ABB RobotStudio station: ABBPingPongRobot.rspag

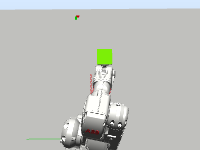
--- station ---
Station ABBPingPongRobot (saved by RobotStudio 6.8.8148.134)
Controller IRB_140_6kg_0.81m
  mechanical unit ROB_1: IRB140_6_81_C_03, 6 joints, base frame (0, 0, 0) mm
Layout (positions relative to the parent item):
  - IRB140_6_81_C_03 [mechanism, from Robots\IRB140_6_81_C_G_03.rslib] at (0, 0, 0) mm; joint values [-0.2001, 0.5892, 0.304, 2.8895, 0.9078, -2.9944] (rad or m)
  - PingPongTool [part] at (563.14, -101.19, 355.17) mm, rotated rx -95.85 ry 89.44 rz -95.98 deg
Attachment: PingPongTool is attached to IRB140_6_81_C_03 / Link6
Targets, tools, work objects and paths stored in the station and not in the controller backup, written as RAPID:
! task T_ROB1
MODULE Module1
  CONST robtarget pHome:=[[200.840292985,299.473805255,-36.431164148],[0.502134661,0.502746249,-0.496734186,0.498359449],[-1,1,-2,0],[9E+09,9E+09,9E+09,9E+09,9E+09,9E+09]];
  CONST robtarget Target_10:=[[200.840292985,299.473805255,-36.431164148],[0.502134661,0.502746249,-0.496734186,0.498359449],[-1,1,-2,0],[9E+09,9E+09,9E+09,9E+09,9E+09,9E+09]];
  PROC PINGPONG()
    ConfL \Off;
    MoveL pPoint,v100,z0,tool0\WObj:=Workobject;
  ENDPROC
ENDMODULE


--- Backups/IRB_140_6kg_0.81m/RAPID/TASK1/PROGMOD/CalibData.mod ---
MODULE CalibData
	TASK PERS wobjdata Workobject:=[FALSE,TRUE,"",[[0,0,0],[1,0,0,0]],[[893.616,92.649,318.739],[0,-0.707106781,0.707106781,0]]];
ENDMODULE

--- Backups/IRB_140_6kg_0.81m/RAPID/TASK1/PROGMOD/Module1.mod ---
MODULE Module1

    VAR num flag:=0;
    VAR bool repeat:=TRUE;
    VAR robtarget pPoint:=[[200.840292985,299.473805255,-36.431164148],[0.502134661,0.502746249,-0.496734186,0.498359449],[-1,1,-2,0],[9E+09,9E+09,9E+09,9E+09,9E+09,9E+09]];
    VAR pos vector;

    PROC Main()

        WHILE flag>-1 DO
            IF flag=1 THEN
                MOVING;
            ENDIF
            WaitTime 0.2;
        ENDWHILE

    ENDPROC

    PROC MOVING()

        ConfL\Off;

        IF repeat THEN
            pPoint:=Offs(pPoint,vector.x,vector.y,0);
            MoveL pPoint,v100,z0,tool0\WObj:=Workobject;
            repeat:=FALSE;
        ENDIF

        flag:=0;
        repeat:=TRUE;

    ENDPROC

ENDMODULE
